{attribute 'Tc2GvlVarNames'}
{attribute 'strict'}
//Tipo Richiesta LGV
TYPE e_Tipo_Richiesta_LGV :
(
	REQ_PRELIEVO_LGV_PIENO	:= 1,	(* Tipo di richiesta LGV = Richiesta di Tipo "PRELIEVO DI ELEMENTO CON MATERIALE" *)
	REQ_DEPOSITO_LGV_PIENO	:= 2,	(* Tipo di richiesta LGV = Richiesta di Tipo "DEPOSITO ELEMENTO CON MATERIALE" *)
	REQ_PRELIEVO_LGV_VUOTO	:= 3,	(* Tipo di richiesta LGV = Richiesta di Tipo "PRELIEVO ELEMENTO SENZA MATERIALE" *)
	REQ_DEPOSITO_LGV_VUOTO	:= 4	(* Tipo di richiesta LGV = Richiesta di Tipo "DEPOSITO ELEMENTO SENZA MATERIALE" *)
	
);
END_TYPE

(* stored: Version 1.1.0.1, ProductVersion 3.1.4024.11
   EnumerationTextList e_Tipo_Richiesta_LGV: Id {c7d2caad-261f-4acf-bbce-0449e8206fd9} *)
